{attribute 'qualified_only'}
VAR_GLOBAL
	Pressure_sensor : INT := 1;
	Pressure_Goal : INT := 1;
END_VAR

(* stored: Version 1.1.0.1, ProductVersion 3.1.4024.12
   GVL GVL: Id {c4b01c67-0cbf-4fd9-b8e9-a595e00bf7a4} *)
